FUNCTION_BLOCK T_StructToJsonFileWriter EXTENDS T_NamedBase
VAR
	filePath : STRING; // fully qualified, including directory
	fileWrite : T_FileWriteBase;
	jDoc : JsonDoc;
	structureName : STRING; // i.e. 'ST_Recipe'
	pointerToStructure : PVOID; // i.e. ADR(recipe)
	sizeOfStructure : UDINT; // i.e. SIZEOF(recipe) 
	jsonWriter : FB_JsonSaxWriter;
	jsonDataTypeWriter : FB_JsonReadWriteDataType;
	_error : BOOL;
	_busy : BOOL;
	_done : BOOL;
END_VAR

fileWrite();
_error S= fileWrite.Error;
_busy := fileWrite.Busy;
_done := fileWrite.Done;

{attribute 'monitoring' := 'call' }
PROPERTY PUBLIC Busy : BOOL
GET
Busy := _busy;
END_GET
END_PROPERTY

{attribute 'monitoring' := 'call' }
PROPERTY PUBLIC Done : BOOL
GET
Done := _done;
END_GET
END_PROPERTY

{attribute 'monitoring' := 'call' }
PROPERTY PUBLIC Error : BOOL
GET
Error := _error;
END_GET
END_PROPERTY

METHOD PUBLIC Reset
fileWrite.ClearWriteBuffer();
jsonWriter.ResetDocument();
_error := FALSE;
LogDebug( 'Reset called' );
END_METHOD

METHOD PUBLIC SetFileParams
VAR_INPUT
	FilePath : Tc2_Utilities.T_MaxString;
	StructureName : STRING; // i.e. 'ST_Recipe'
	PointerToStructure : PVOID; // i.e. ADR(recipe) 
	SizeOfStructure : UDINT; // i.e. SIZEOF(recipe) 
END_VAR
THIS^.filePath := FilePath; // for debug only.
fileWrite.SetFilePath(FilePath := FilePath);

THIS^.structureName := StructureName;
THIS^.pointerToStructure := PointerToStructure; 
THIS^.sizeOfStructure := SizeOfStructure;
END_METHOD

METHOD PUBLIC WriteToFile // Attempt to write structure to file
VAR
	docSize : UDINT;
END_VAR
IF _error THEN
	LogError ( 'Cannot write to file while block is in an error state. Reset first' );
	RETURN;
	
END_IF

jsonWriter.ResetDocument();

_error S= NOT jsonDataTypeWriter.AddJsonValueFromSymbol(
						fbWriter := jsonWriter,
						sDatatype := structureName,
						nData := sizeOfStructure,
						pData := pointerToStructure	
					);
				
IF _error THEN
	LogError ( 'Error while creating json file from structure. Check argument for SetFileParams' );
	RETURN;
	
END_IF

docSize := jsonWriter.CopyDocument(
					pDoc := jDoc,
					nDoc := SIZEOF( jDoc )
				);

fileWrite.ClearWriteBuffer();

_error S= NOT fileWrite.AppendToBuffer(
						pDataForBuffer := ADR( jdoc ),
						DataLength := docSize
					);

IF _error THEN
	LogError ( 'Error while adding to write buffer. Try increasing JsonDoc size using JsonParams in library, or TC mailbox size.' );
	RETURN;
	
END_IF		
			
_error S= NOT fileWrite.StartWrite();

IF _error THEN
	LogError ( 'Error  starting file write. Try calling Reset first.' );
	RETURN;
	
END_IF
END_METHOD

END_FUNCTION_BLOCK

(* stored: Version 1.1.0.1, ProductVersion 3.1.4022.18
   POU T_StructToJsonFileWriter: Id {fd59d0dd-3f9a-096c-1145-5dd2bb026d0f}, SpecialFunc None
   Property Busy: Id {1850d0b4-67f1-0956-388d-78848d7d1e7e}
   Get Get: Id {2665f752-0177-0ced-2048-525d127bc931}
   Property Done: Id {1bb13495-e23b-063e-04bc-28359a31cd2a}
   Get Get: Id {7b67d981-310f-09fd-1269-613ba87d81b6}
   Property Error: Id {640531db-ca33-03e3-08a6-c5eeaf8bf680}
   Get Get: Id {5830fbc2-b56e-027e-15d2-c0cca378a073}
   Method Reset: Id {06d5ff98-34b0-0099-10c5-d3a840205290}
   Method SetFileParams: Id {7a8b72e9-c6b3-01da-10b6-970addc33cca}
   Method WriteToFile: Id {2a0ecc25-7db0-06f7-3c64-41521e99da6c} *)
